// Standalone logger, if no logger is attached to FB_Event, nice for tessting
FUNCTION F_Log : BOOL
VAR_INPUT
	fbMessage:			REFERENCE TO FB_Message;
END_VAR
VAR
	sMessage:			STRING(255):= 'Logger = 0 | ';
    nIndex:				UINT;
END_VAR
(*
    Tc3_Event – TwinCAT 3 Event Logging Framework
    Copyright (c) Peter Zerlauth

    This component is provided under a Dual Licensing Model:

    1. GPLv3 Open-Source License
       - Free for personal, educational, and non-commercial use.
       - Commercial use allowed only if the entire application is published
         under GPLv3, including all modifications to this code.
       - Requires full disclosure of source code for derivative works.

    2. Commercial License
       - Required for integration into proprietary or closed-source products.
       - Removes all GPLv3 copyleft obligations.
       - Includes optional warranty, professional support, and long-term
         maintenance options.

    For commercial licensing, contact:
        info@peterzerlauth.com

    By using this Function Block you agree to the terms of the selected license.
*)

// --- Build log line
sMessage:= CONCAT('Logger null | ', fbMessage.sSource);
sMessage:= CONCAT(sMessage, ': ');
sMessage:= CONCAT(sMessage, fbMessage.sDefault);

// --- Keep active
IF F_Filter(fbMessage) THEN 
	RETURN;
END_IF

// --- Add to buffer ---
IF GVL.nBuffer < 99 THEN
    GVL.aBuffer[GVL.nBuffer]:= fbMessage;
    GVL.aBuffer[GVL.nBuffer].nTimestamp := GVL.nTimestamp;
    GVL.nBuffer := GVL.nBuffer + 1;
END_IF

// --- Log message ---
CASE fbMessage.eLogLevel OF
    E_LogLevel.Verbose, E_LogLevel.Info:
        ADSLOGSTR(ADSLOG_MSGTYPE_HINT, '%s', sMessage);
    E_LogLevel.Warning:
        ADSLOGSTR(ADSLOG_MSGTYPE_WARN, '%s', sMessage);
    E_LogLevel.Error, E_LogLevel.Critical:
        ADSLOGSTR(ADSLOG_MSGTYPE_ERROR, '%s', sMessage);
END_CASE

// --- Remove outdated messages
F_Remove();

F_Log := TRUE;

END_FUNCTION

(* stored: Version 1.1.0.1
   POU F_Log: Id {3d8b8d8d-2aeb-485f-a382-76004536aaec}, SpecialFunc None *)
